{attribute addProperty BoxType "EL2034-0000-0016"}
{attribute addProperty Id "DiagAT %I*ARRAY[0..3] OF Diag_4CD4E3A23240ChannelAT %Q*ARRAY[0..3] OF Channel_7F374EB03240WcStateAT %I*WcState_F855686C1620InfoDataAT %I*InfoData_192954DE1620"}
{attribute addProperty CRC "2677586100"}
{attribute addProperty SizeInBites "96"}
{attribute addProperty SizeInBytes "12"}
TYPE EL2034_79951597 :
STRUCT
	{attribute addProperty Name "Diag"}
	Diag : ARRAY[0..3] OF Diag_4CD4E3A2;
	{attribute addProperty Name "Channel"}
	Channel : ARRAY[0..3] OF Channel_7F374EB0;
	{attribute addProperty Name "WcState"}
	WcState : WcState_F855686C;
	{attribute addProperty Name "InfoData"}
	InfoData : InfoData_192954DE;
END_STRUCT
END_TYPE

(* stored: Version 1.2.0.0, ProductVersion 3.1.4024.9
   DUT EL2034_79951597: Id {eae7b7ec-d961-4dcc-8b78-9dffe787a6d5} *)
